TYPE STM_Control_Control :
STRUCT
	Enable : BIT;
	Reset : BIT;
	ReduceTorque : BIT;
	
	{attribute 'hide'}
	padding_0_3	: BIT;
	{attribute 'hide'}
	padding_0_4	: BIT;
	{attribute 'hide'}
	padding_0_5	: BIT;
	{attribute 'hide'}
	padding_0_6	: BIT;
	{attribute 'hide'}
	padding_0_7	: BIT;
	{attribute 'hide'}
	padding_1_0	: BIT;
	{attribute 'hide'}
	padding_1_1	: BIT;
	{attribute 'hide'}
	padding_1_2	: BIT;
	{attribute 'hide'}
	padding_1_3	: BIT;
	{attribute 'hide'}
	padding_1_4	: BIT;
	{attribute 'hide'}
	padding_1_5	: BIT;	
	{attribute 'hide'}
	padding_1_6	: BIT;
	{attribute 'hide'}
	padding_1_7	: BIT;
END_STRUCT
END_TYPE

(* stored: Version 1.1.0.1, ProductVersion 3.1.4024.3
   DUT STM_Control_Control: Id {38d95f56-9a67-4239-9a60-32474cd98971} *)
